(* PLC project poST.project, poSTIDE *)
(* stored: creationDateTime 2021-08-31T00:00:00.000000 *)

FUNCTION SUB_TOD_TIME : TIME_OF_DAY
  VAR_INPUT
    in1 : TIME_OF_DAY;
    in2 : TIME;
  END_VAR

END_FUNCTION
